SUBAPPLICATION Uebung_003b2_sub (* IX auf QX (generisch) *)
  (* Standard: 61499-2; Description: Copyright (c) 2023 Meisterschulen am Ostbahnhof This program and the accompanying materials are made available under the terms of the Eclipse Public License 2.0 which is available at https://www.eclipse.org/legal/epl-2.0/ SPDX-License-Identifier: EPL-2.0 *)
  (* Version 1.0, 2023-10-23, Franz Höpfinger, Meisterschulen am Ostbahnhof *)
  PACKAGE Uebungen;
  IMPORT DataPanel::io::MI::DQ::DataPanel_MI_DO_S;
  IMPORT DataPanel::io::MI::const::MI;
  IMPORT Funk::io::DI::Funk_DI;
  IMPORT Funk::io::DI::Funk_DI_S;
  IMPORT DataPanel::io::MI::DQ::DataPanel_MI_DO::Invalid;
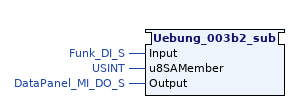
  VAR_INPUT
    Input : Funk::io::DI::Funk_DI_S := Funk_DI::Invalid; (* Identify the Input DigitalInput_Key_01 etc.. *)
    u8SAMember : USINT := MI::MI_00; (* Node SA 224..239 *)
    Output : DataPanel::io::MI::DQ::DataPanel_MI_DO_S := Invalid; (* Identify the Output DigitalOutput_1A..8B and Input_Power_Port_5..8 *)
  END_VAR
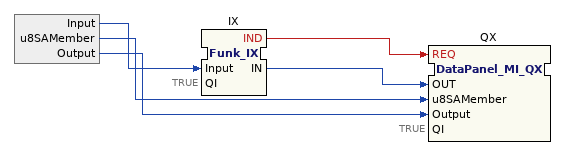
  FBS
    QX : DataPanel::io::MI::DQ::DataPanel_MI_QX(QI := TRUE);
    IX : Funk::io::DI::Funk_IX(QI := TRUE);
  END_FBS
  EVENT_CONNECTIONS
    IX.IND TO QX.REQ;
  END_CONNECTIONS
  DATA_CONNECTIONS
    IX.IN TO QX.OUT;
    Input TO IX.Input;
    u8SAMember TO QX.u8SAMember;
    Output TO QX.Output;
  END_CONNECTIONS
END_SUBAPPLICATION
